{attribute 'linkalways'} 
{attribute 'no_explicit_call' := 'This FB is a CLASS and must be accessed using methods or properties'}
{attribute 'enable_dynamic_creation'}
FUNCTION_BLOCK ABSTRACT EnumDatatypeBase EXTENDS UserDefinedDatatypeBase IMPLEMENTS I_EnumDatatype
VAR
	_baseType : I_Datatype;
	enumerations : Dictionary;
END_VAR

METHOD PROTECTED AddBaseType
VAR_INPUT
	BaseType : I_Datatype;
END_VAR
_baseType := BaseType;
END_METHOD

METHOD PROTECTED AddEnumeration
VAR_INPUT
	Enumeration : T_MAXSTRING;
	Value : ANY;
END_VAR
enumerations.AddOrUpdate(Enumeration, Value);
END_METHOD

METHOD PRIVATE CreateEnumError : I_Error
VAR_INPUT
	Enum : T_MAXSTRING;
END_VAR
VAR
	pError : POINTER TO UnknownEnumerationError;
END_VAR
pError := __NEW(UnknownEnumerationError(EnumString := Enum));
CreateEnumError := pError^;
END_METHOD

PROPERTY PUBLIC Datatype : T_MAXSTRING
GET
Datatype := 'ENUM';
END_GET
END_PROPERTY

METHOD ABSTRACT IsEnumeratorValueEqual : BOOL
VAR_INPUT
	Enumerator : I_KeyValueForwardEnumerator;
END_VAR
END_METHOD

METHOD PROTECTED OnSerializeTypeWith
VAR_INPUT
	Serializer : I_Serializer;
END_VAR
SUPER^.OnSerializeTypeWith(Serializer);
SerializeEnums(Serializer);
SerializeBaseType(Serializer);
END_METHOD

METHOD PRIVATE SerializeBaseType
VAR_INPUT
	Serializer : I_Serializer;
END_VAR
IF _baseType = 0 THEN
	RETURN;
END_IF

Serializer.AddKey('baseType');
_baseType.SerializeTypeWith(Serializer);
END_METHOD

METHOD PRIVATE SerializeEnums
VAR_INPUT
	Serializer : I_Serializer;
END_VAR
VAR
	enumerator : I_KeyValueForwardEnumerator;
END_VAR
Serializer.AddKey('enumerations');
Serializer.StartArray();

enumerator := enumerations.GetKeyValueEnumerator();

WHILE enumerator.MoveNext() DO
	Serializer.AddString(enumerator.Key);
END_WHILE

enumerator.Dispose();

Serializer.EndArray();
END_METHOD

METHOD PUBLIC SerializeWith
VAR_INPUT
	Serializer : I_Serializer;
END_VAR
VAR
	returnKey : T_MAXSTRING;
	enumerator : I_KeyValueForwardEnumerator;
END_VAR
enumerator := enumerations.GetKeyValueEnumerator();
returnKey := 'UNDEFINED';

WHILE (enumerator.MoveNext()) DO
	
	IF IsEnumeratorValueEqual(enumerator) THEN
		returnKey := enumerator.key;
		EXIT;
	END_IF

END_WHILE

Serializer.AddString(returnKey);
enumerator.Dispose();
END_METHOD

METHOD TryDeserializeFrom : BOOL
VAR_INPUT
	Deserializer : I_Deserializer;
	Feedback : I_DeserializerFeedback;
END_VAR
VAR
	key : T_MAXSTRING;
	error : I_Error;
END_VAR
IF NOT Deserializer.TryGetString(key, Feedback) THEN
	RETURN;
END_IF

IF NOT enumerations.TryGetValueTo(key, Address, Size) THEN
	error := CreateEnumError(key);
	Feedback.LogError(error);
	RETURN;
END_IF
END_METHOD

METHOD PUBLIC TryResolveAsEnumType : BOOL
VAR_INPUT
	Destination : REFERENCE TO I_EnumDatatype;
END_VAR
Destination := THIS^;
TryResolveAsEnumType := TRUE;
END_METHOD

END_FUNCTION_BLOCK

(* stored: Version 1.1.0.1, ProductVersion 3.1.4024.12
   POU EnumDatatypeBase: Id {b7a95de7-b421-0e8f-2327-fed6e5aa41c9}, SpecialFunc None
   Folder Private: Id {abe5b4bb-f5fe-0010-0885-5bc659c7d995}
   Folder Protected: Id {df80dcfd-7e83-0e16-3e74-a8452c92beda}
   Method AddBaseType: Id {5697f491-86c4-02ef-188a-e14d3091e797}
   Method AddEnumeration: Id {6ce4bf04-6cb4-0cfb-3763-a52d39a150e4}
   Method CreateEnumError: Id {e4129c80-b976-0890-3706-5b891a6f721e}
   Property Datatype: Id {526e7ac1-93e0-0467-3a70-e27a408f2f7c}
   Get Get: Id {3eed1a3c-d9b3-0f10-1751-427e0097a390}
   Method IsEnumeratorValueEqual: Id {f88c9827-7762-0230-3ec6-56ecb680df4b}
   Method OnSerializeTypeWith: Id {3864821e-09dc-0d14-2436-07a6354a045b}
   Method SerializeBaseType: Id {f93acaf6-72b8-0a12-374c-417568457829}
   Method SerializeEnums: Id {2167f6be-7212-014b-0780-288bef4900ce}
   Method SerializeWith: Id {ddbc34c4-cbd6-0ef0-22ff-c527be90a527}
   Method TryDeserializeFrom: Id {d8fbce8c-ee8b-052e-1578-7e5cd0c5b33a}
   Method TryResolveAsEnumType: Id {7fff9ffe-4f82-0d07-1232-c7244381b275} *)
